FUNCTION_BLOCK SAFE_MUL_4 (* Calculate arithmetical product of numeric inputs, saturating on overflow (generic FB) *)
  (* Standard: 61131-3; Classification: saturating arithmetic function; Description: Copyright (c) 2026 HR Agrartechnik GmbH This program and the accompanying materials are made available under the terms of the Eclipse Public License 2.0 which is available at https://www.eclipse.org/legal/epl-2.0/ SPDX-License-Identifier: EPL-2.0 *)
  (* Version 1.0, 2026-08-27, Franz Höpfinger, HR Agrartechnik GmbH, initial API and implementation and/or initial documentation *)
  PACKAGE SafeArithmetic::arithmetic;
  {SET_ATTRIBUTE(eclipse4diac::core::GenericClassName, 'GEN_SAFE_MUL')}
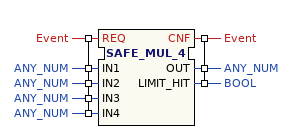
  EVENT_INPUT
    REQ WITH IN1, IN2, IN3, IN4; (* Normal Execution Request *)
  END_EVENT
  EVENT_OUTPUT
    CNF WITH OUT, LIMIT_HIT; (* Execution Confirmation *)
  END_EVENT
  VAR_INPUT
    IN1 : ANY_NUM; (* first factor *)
    IN2 : ANY_NUM; (* second factor *)
    IN3 : ANY_NUM; (* third factor *)
    IN4 : ANY_NUM; (* fourth factor *)
  END_VAR
  VAR_OUTPUT
    OUT : ANY_NUM; (* MUL result, clamped to the valid range of the result type *)
    LIMIT_HIT : BOOL; (* TRUE if the result was clamped due to overflow *)
  END_VAR
END_FUNCTION_BLOCK
